FUNCTION_BLOCK FB_WinchInterface
VAR_INPUT
	enable : BOOL := FALSE;
	reset : BOOL := FALSE;
	stopp : BOOL := FALSE;
	
	mode : UINT := 0;
	control : ST_ControlWinch;

	
END_VAR
VAR_OUTPUT
	active : BOOL := FALSE;
	
	feedback : ST_FeedbackWinch;
	
	testL : LREAL := 0.7;
END_VAR
VAR
	// HMI feedback	
	pTxHmi : POINTER TO ST_TxHmiWinch;
	
	// MC2 Functions
	axis : AXIS_REF;
	fbPower : MC_Power;
	fbReset : MC_Reset;
	fbExtSetPointGenEnable : MC_ExtSetPointGenEnable;
	fbExtSetPointGenDisable : MC_ExtSetPointGenDisable;
	fbReadParameterSet : MC_ReadParameterSet;
	stAxisParameterSet : ST_AxisParameterSet;
	
	// Setpoint generation
	timer : TON;
	
	Ts : LREAL := 0.005;
	
	omega : LREAL := 1.0;
	beta : LREAL := 1.0;
	
	
	l : LREAL := 0.0;
	l_t : LREAL := 0.0;
	l_tt : LREAL := 0.0;
	direction : DINT := 0;
	
	
	// Physical wire length conversion factors
	
	
END_VAR

// Update axis data
axis();

// Return feedback data
feedback.l := (7600.0 - LREAL_TO_REAL(axis.NcToPlc.ActPos) + 626.0)/1000.0;
feedback.l_t := -LREAL_TO_REAL(axis.NcToPlc.ActVelo)/1000.0;
feedback.l_tt := -LREAL_TO_REAL(axis.NcToPlc.ActAcc)/1000.0;


// Read parameter set
fbReadParameterSet(
	Axis := axis,
	Parameter := stAxisParameterSet,
	Execute := FALSE
);
fbReadParameterSet(
	Axis := axis,
	Parameter := stAxisParameterSet,
	Execute := TRUE
);

// Check operation mode
IF fbPower.Status THEN
	CASE mode OF
	0 : 
		// Settled
		omega := 1.0;
		
		// Disable external setpoint when generator is close to standstill!
		IF ABS(l_t) < 1.0 AND ABS(l_tt) < 0.1 THEN
			DisableExtSetPoint();
		END_IF
	1 : 
		// Enagaged
		omega := 1.0;

		// Enable external setpoint
		EnableExtSetPoint();
	2 : 
		// Enagaged - Fast
		omega := 10.0;
		
		// Enable external setpoint
		EnableExtSetPoint();
	ELSE
		// Return to settled if wrong mode is set!
		mode := 0;
	END_CASE
END_IF

// Generate Trqajectory
GenerateTrajectory();

// Feed extrenal setpoints to axis interface
MC_ExtSetPointGenFeed(
	Axis := axis,
	Position := l,
	Velocity := l_t,
	Acceleration := l_tt,
	Direction := direction
);

// Set power status for winch
IF enable THEN
	// Power on the drive
	fbPower(
		Axis := axis,
		Enable := TRUE,
		Enable_Positive := TRUE,
		Enable_Negative := TRUE
	);
	// Rest disable
	reset := FALSE;
ELSE
	mode := 0;
	IF NOT fbExtSetPointGenDisable.Busy AND fbExtSetPointGenDisable.Done THEN
		// Power off the drive
		fbPower(
			Axis := axis,
			Enable := FALSE,
			Enable_Positive := FALSE,
			Enable_Negative := FALSE
		);
	END_IF
END_IF

METHOD PRIVATE DisableExtSetPoint : BOOL
VAR_INPUT
END_VAR
fbExtSetPointGenDisable(
	Axis := axis,
	Execute := TRUE
);
fbExtSetPointGenEnable(
	Axis := axis,
	Execute := FALSE
);
END_METHOD

METHOD PRIVATE EnableExtSetPoint : BOOL
VAR_INPUT
END_VAR
fbExtSetPointGenDisable(
	Axis := axis,
	Execute := FALSE
);
fbExtSetPointGenEnable(
	Axis := axis,
	Execute := TRUE
);
END_METHOD

METHOD FB_init : BOOL
VAR_INPUT
	bInitRetains : BOOL; // if TRUE, the retain variables are initialized (warm start / cold start)
	bInCopyCode : BOOL;  // if TRUE, the instance afterwards gets moved into the copy code (online change)
	
	// Init variables
	_pTxHmi : POINTER TO ST_TxHmiStewart;
END_VAR
// Ensure Power of axis is disbaled at startup
fbPower(
	Axis := axis,
	Enable := FALSE,
	Enable_Positive := FALSE,
	Enable_Negative := FALSE
);

fbExtSetPointGenDisable(
	Axis := axis,
	Execute := FALSE
);
fbExtSetPointGenEnable(
	Axis := axis,
	Execute := FALSE
);
END_METHOD

METHOD PRIVATE GenerateTrajectory : BOOL
VAR_INPUT
END_VAR

VAR
	// Setpoints
	pos : LREAL;
	vel : LREAL;
	acc : LREAL;
END_VAR
IF mode = 0 THEN
	// Settle in last position
	pos := axis.NcToPlc.ActPos;
	vel := 0.0;
	acc := 0.0;
ELSE
	// Follow input trajectory
	pos := 7600.0 + 626.0 - REAL_TO_LREAL(control.l)*1000.0;
	vel := -REAL_TO_LREAL(control.l_t)*1000.0;
	acc := -REAL_TO_LREAL(control.l_tt)*1000.0;
END_IF

// Generate trajectory using trajectory filter
l_tt := acc + 2*beta*omega*(vel - l_t) + omega*omega*(pos - l);
l_t := l_t + l_tt*Ts;
l := l + l_t*Ts;

// Set setpoint direction
IF l_t = 0.0 AND l_tt = 0.0 THEN
	// Standstill
	direction := 0;
ELSIF l_t >= 0.0 THEN
	// Positive motion
	direction := 1;
ELSE
	// Negative motion
	direction := -1;
END_IF
END_METHOD

METHOD PRIVATE UpdateHMI : BOOL
VAR_INPUT
END_VAR
// Update HMI variables
END_METHOD

END_FUNCTION_BLOCK

(* stored: Version 1.1.0.1, ProductVersion 3.1.4022.7
   POU FB_WinchInterface: Id {04fd987b-6b6d-4a7c-b1e1-6e43123e7fac}, SpecialFunc None
   Method DisableExtSetPoint: Id {8625365a-3f23-4e76-ba3a-d36439744fe2}
   Method EnableExtSetPoint: Id {d86b78de-9d3a-4053-bd82-f21f9d22062b}
   Method FB_init: Id {4ef8ab5f-4b43-4ec7-898b-623c39afb859}
   Method GenerateTrajectory: Id {a2b9dbe1-8750-44c6-b8bf-0dc16aa5e2fd}
   Method UpdateHMI: Id {66797478-8570-421d-ad5d-4d9d457815e9} *)
